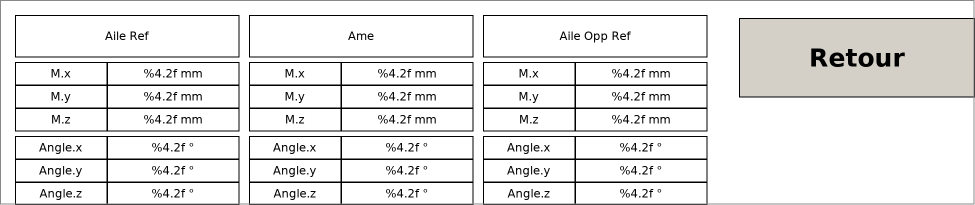
VISUALIZATION Chgt_Reperes  // 975x205
    Rectangle (15,15 224x42), "Aile Ref"
    Rectangle (15,62 92x23), "M.x"
    Rectangle (107,62 132x23), "%4.2f mm", text variable: Palpage_laser.M[1].X
    Rectangle (15,85 92x23), "M.y"
    Rectangle (107,85 132x23), "%4.2f mm", text variable: Palpage_laser.M[1].Y
    Rectangle (15,108 92x23), "M.z"
    Rectangle (107,108 132x23), "%4.2f mm", text variable: Palpage_laser.M[1].Z
    Rectangle (15,136 92x23), "Angle.x"
    Rectangle (107,136 132x23), "%4.2f °", text variable: Palpage_laser.Angles_Rotation[1].X
    Rectangle (15,159 92x23), "Angle.y"
    Rectangle (107,159 132x23), "%4.2f °", text variable: Palpage_laser.Angles_Rotation[1].Y
    Rectangle (15,182 92x23), "Angle.z"
    Rectangle (107,182 132x23), "%4.2f °", text variable: Palpage_laser.Angles_Rotation[1].Z
    Rectangle (249,15 224x42), "Ame"
    Rectangle (249,62 92x23), "M.x"
    Rectangle (341,62 132x23), "%4.2f mm", text variable: Palpage_laser.M[2].X
    Rectangle (249,85 92x23), "M.y"
    Rectangle (341,85 132x23), "%4.2f mm", text variable: Palpage_laser.M[2].Y
    Rectangle (249,108 92x23), "M.z"
    Rectangle (341,108 132x23), "%4.2f mm", text variable: Palpage_laser.M[2].Z
    Rectangle (249,136 92x23), "Angle.x"
    Rectangle (341,136 132x23), "%4.2f °", text variable: Palpage_laser.Angles_Rotation[2].X
    Rectangle (249,159 92x23), "Angle.y"
    Rectangle (341,159 132x23), "%4.2f °", text variable: Palpage_laser.Angles_Rotation[2].Y
    Rectangle (249,182 92x23), "Angle.z"
    Rectangle (341,182 132x23), "%4.2f °", text variable: Palpage_laser.Angles_Rotation[2].Z
    Rectangle (483,15 224x42), "Aile Opp Ref"
    Rectangle (483,62 92x23), "M.x"
    Rectangle (575,62 132x23), "%4.2f mm", text variable: Palpage_laser.M[3].X
    Rectangle (483,85 92x23), "M.y"
    Rectangle (575,85 132x23), "%4.2f mm", text variable: Palpage_laser.M[3].Y
    Rectangle (483,108 92x23), "M.z"
    Rectangle (575,108 132x23), "%4.2f mm", text variable: Palpage_laser.M[3].Z
    Rectangle (483,136 92x23), "Angle.x"
    Rectangle (575,136 132x23), "%4.2f °", text variable: Palpage_laser.Angles_Rotation[3].X
    Rectangle (483,159 92x23), "Angle.y"
    Rectangle (575,159 132x23), "%4.2f °", text variable: Palpage_laser.Angles_Rotation[3].Y
    Rectangle (483,182 92x23), "Angle.z"
    Rectangle (575,182 132x23), "%4.2f °", text variable: Palpage_laser.Angles_Rotation[3].Z
    Rectangle (739,18 236x79), "Retour"
        OnMouseClick: change screen: MenuPrincipal
END_VISUALIZATION

(* stored: Version 1.1.0.1
   Visu Chgt_Reperes: Id {2bace917-3852-40bc-b38a-f2e8423626ea} *)
